PROGRAM PsdBkgrdSerialCom
VAR_INPUT
	Config : PsdConfig;
END_VAR
VAR
END_VAR

// ScreensConfigs
IF Config.ScreenConfigs.DM430GNScreenConfigFS.IsEnabled THEN
	BkgrdSerialScreenFS();
END_IF
IF Config.ScreenConfigs.DM430GNScreenConfigBS.IsEnabled THEN
	BkgrdSerialScreenBS();
END_IF

END_PROGRAM

(* stored: Version 1.1.0.1, ProductVersion 3.1.4024.12
   POU PsdBkgrdSerialCom: Id {afb62224-d23e-49ab-a16e-8c18a0a03443}, SpecialFunc None *)
